FUNCTION_BLOCK FB_Observer_ULINT EXTENDS FB_AbstractObserver
VAR
    _nVal:              ULINT;
END_VAR

METHOD FB_init : BOOL
VAR_INPUT
	bInitRetains : BOOL; // if TRUE, the retain variables are initialized (warm start / cold start)
	bInCopyCode : BOOL;  // if TRUE, the instance afterwards gets moved into the copy code (online change)
END_VAR
THIS^._nTypeClass := __SYSTEM.TYPE_CLASS.TYPE_ULINT;
THIS^._pVal := ADR(THIS^._nVal);
THIS^._nSize := SIZEOF(THIS^._nVal);
END_METHOD

PROPERTY nValue64 : ULINT
GET
nValue64 := THIS^._nVal;
END_GET
END_PROPERTY

END_FUNCTION_BLOCK

(* stored: Version 1.1.0.1, ProductVersion 3.1.4024.12
   POU FB_Observer_ULINT: Id {824a1673-2aeb-0640-0a92-6fb92ce1a64d}, SpecialFunc None
   Method FB_init: Id {3beba01c-12a7-00b2-31aa-10f8eae14b74}
   Property nValue64: Id {e4fccded-9aaa-03cc-16c9-873e6f32628b}
   Get Get: Id {4bc01161-7215-0490-3c8c-4608e232d494} *)
